SUBAPPLICATION Uebung_120x_sub (* Subapplication Type *)
  (* Standard: 61499-2 *)
  (* Version 1.0, 2025-10-22, Franz Höpfinger, Meisterschulen am Ostbahnhof, initial API and implementation and/or initial documentation *)
  PACKAGE Uebungen;
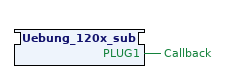
  PLUGS
    PLUG1 : isobus::pgn::tx::Callback;
  END_PLUGS
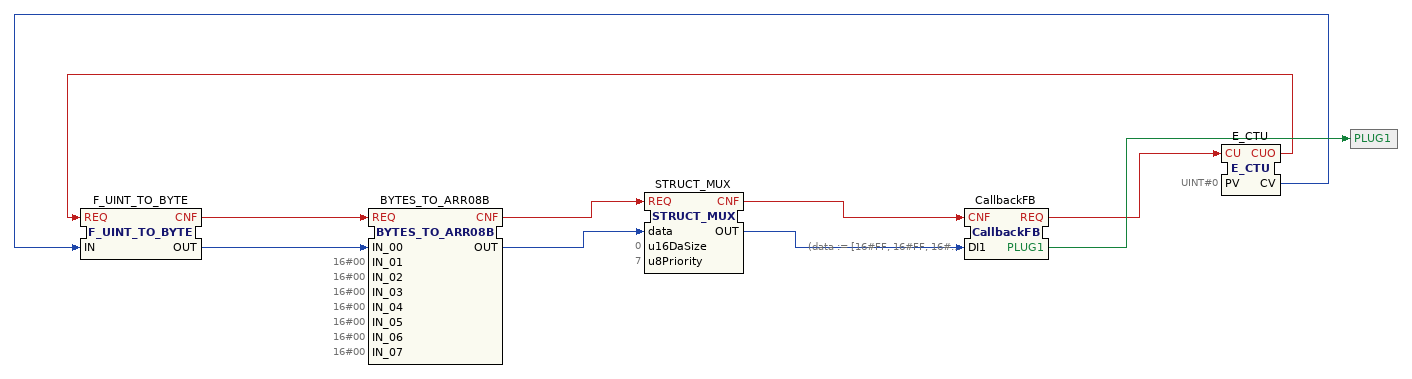
  FBS
    CallbackFB : isobus::pgn::tx::CallbackFB(DI1 := (data := [16#FF, 16#FF, 16#FF, 16#FF, 16#FF, 16#FF, 16#FF, 16#FF]));
    E_CTU : iec61499::events::E_CTU(PV := UINT#0);
    STRUCT_MUX : eclipse4diac::convert::STRUCT_MUX(u16DaSize := 0, u8Priority := 7); {SET_ATTRIBUTE(StructuredType, isobus::pgn::CAN_MSG)}
    BYTES_TO_ARR08B : logiBUS::utils::conversion::arr::reversing::BYTES_TO_ARR08B(IN_01 := 16#00, IN_02 := 16#00, IN_03 := 16#00, IN_04 := 16#00, IN_05 := 16#00, IN_06 := 16#00, IN_07 := 16#00);
    F_UINT_TO_BYTE : iec61131::conversion::F_UINT_TO_BYTE;
  END_FBS
  EVENT_CONNECTIONS
    CallbackFB.REQ TO E_CTU.CU;
    STRUCT_MUX.CNF TO CallbackFB.CNF;
    BYTES_TO_ARR08B.CNF TO STRUCT_MUX.REQ;
    F_UINT_TO_BYTE.CNF TO BYTES_TO_ARR08B.REQ;
    E_CTU.CUO TO F_UINT_TO_BYTE.REQ;
  END_CONNECTIONS
  DATA_CONNECTIONS
    STRUCT_MUX.OUT TO CallbackFB.DI1;
    BYTES_TO_ARR08B.OUT TO STRUCT_MUX.data;
    F_UINT_TO_BYTE.OUT TO BYTES_TO_ARR08B.IN_00;
    E_CTU.CV TO F_UINT_TO_BYTE.IN;
  END_CONNECTIONS
  ADAPTER_CONNECTIONS
    CallbackFB.PLUG1 TO PLUG1;
  END_CONNECTIONS
END_SUBAPPLICATION
